Fanuc KAREL source: IO0099.KL

PROGRAM IO0099
%STACKSIZE=65535
%PRIORITY=65535
%NOLOCKGROUP
ROUTINE RTEST FROM IO0099
ROUTINE RTEST
VAR
L1 : ARRAY[3] OF INTEGER
L2 : XYZWPR
L3 : JOINTPOS9
L4 : POSITION
S1 : INTEGER
U2C_38 : REAL
U2C_39 : REAL
U2C_40 : BOOLEAN
U2C_41 : REAL
BEGIN
S1=1
L1[1]=2
U2C_40=TRUE
U2C_41=1.0
-- UNSAFE_SOURCE_IR line 19: IF (native_io_value(8, 17) = 1) THEN
S1=(S1 + 1)
ENDIF
END RTEST
BEGIN
RTEST
END IO0099
